Staubli VAL3: start.pgx

program start()
  local num l_nFbkPeriod
  local num l_nMotionPeriod
  local num l_nTrajPeriod
  local num l_nScreenUpdate
  local string l_sVersionMajor
  local num l_nVersionMajor
  local bool l_bOkMajor
  local string l_sVersionMinor
  local num l_nVersionMinor
  local bool l_bOkMinor
begin
  // Copyright (c) 2016, Ocado Technology - Robotics Research Team
  //
  // Licensed under the Apache License, Version 2.0 (the "License");
  // you may not use this file except in compliance with the License.
  // You may obtain a copy of the License at
  //
  //     http://www.apache.org/licenses/LICENSE-2.0
  //
  // Unless required by applicable law or agreed to in writing, software
  // distributed under the License is distributed on an "AS IS" BASIS,
  // WITHOUT WARRANTIES OR CONDITIONS OF ANY KIND, either express or implied.
  // See the License for the specific language governing permissions and
  // limitations under the License.


  // Load interface library for CS8 or CS9
  //
  // CS9 handles the UI differently than CS8, requires
  // the UI funtions to be loaded in seperate libraries

  if(mid(getVersion("System"),1,1) == "7")
    // CS8 - VAL 3 rev 7
    // Check for VAL 3 version >= 7.7
    l_sVersionMajor = mid(getVersion("VAL3"),1,1)
    l_sVersionMinor = mid(getVersion("VAL3"),2,1)
    toNum(l_sVersionMajor, l_nVersionMajor, l_bOkMajor)
    toNum(l_sVersionMinor, l_nVersionMinor, l_bOkMinor)
    if(!l_bOkMajor or !l_bOkMinor)
      popUpMsg("Error reading VAL 3 version")
      taskKill("ros_server~")
    endIf
    if( !((l_nVersionMajor == 7) and (l_nVersionMinor >= 7)))
      // VAL 3 version is too old
      popUpMsg("Error: VAL 3 version is < 7.7, socket communication will not work!")
      taskKill("ros_server~")
    endIf
    libInterface:libLoad("ros_libs/UserInterface/interfaceCS8")
  elseIf(mid(getVersion("System"),1,1) == "8")
    // CS9 - VAL 3 rev 8
    libInterface:libLoad("ros_libs/UserInterface/interfaceCS9")
  endIf

  // feedback task will run every 20ms (50Hz)
  l_nFbkPeriod=0.02
  //l_nFbkPeriod = 0.032 // 30Hz
  //l_nFbkPeriod = 0.05  // 20Hz
  //l_nFbkPeriod = 1.0   //  1Hz

  // motion control task will run every 4ms (250Hz)
  l_nMotionPeriod = 0.004
  //l_nMotionPeriod=0.012  // 83Hz
  //l_nMotionPeriod = 0.05 // 20Hz

  // data (trajectory) reception task will run every 4ms (250Hz)
  l_nTrajPeriod = 0.004
  // not in use at the moment
  l_nScreenUpdate = 1.0

  sStreamTaskName = "streamerTask"
  sTrajPtTaskName = "trajPtTask"
  sMotionTaskName = "motionTask"
  sScreenTaskName = "screenTask"
  sHtbtTaskName = "htbtTask"
  sSystemTaskName = "systemTask"

  // initialise TCP/IP parameters
  call initParams()
  // setup prefix and header of ROS messages
  call setupRosMsgs()

  // socket connection status flags: initially disconnected
  nInConnFlag = 0
  nOutConnFlag = 0
  nSystemConnFlag = 0

  // flag defining whether velocity to be overwritten to max. vel.
  bOverwriteVel = false

  nPtsPopped = 0
  nMovePts = 0

  // flush buffer of incoming socket
  clearBuffer(siTcpIpMotion)
  // flush buffer of outgoing socket
  clearBuffer(siTcpIpFbk)
  // flush buffer of system request socket
  clearBuffer(siTcpIpSystem)

  // check if robot is not in emergency stop and wait until estop is reset
  if(esStatus() == 2)
    popUpMsg("Please reset E-Stop")
    wait(esStatus() < 2)
  endIf

  // before anything else, enable power (only works if robot is in remote mode)
  if(!isPowered())
    if(workingMode() >= 4)
      do
        enablePower()
        delay(2)
      until isPowered()
    else
      popUpMsg("Power must be enabled manually")
    endIf
  endIf

  // reset motion, potentially setting a start joint position for calling autoConnect() in the future
  resetMotion()

  // create joint state and robot status streamer task to send data to industrial_robot_client
  taskCreateSync sStreamTaskName, l_nFbkPeriod, bFbkOverrun, dataStreamer()

  // create trajectory point task to receive data from industrial_robot_client
  taskCreateSync sTrajPtTaskName, l_nTrajPeriod, bTrajPtOverrun, dataReceiver()
  //taskCreate sTrajPtTaskName, 100, dataReceiver()

  // create motion task to synchronously apply motion commands to robot
  taskCreateSync sMotionTaskName, l_nMotionPeriod, bMotionOverrun, motionControl()

  // create synchronous task to update screen
  //taskCreateSync sScreenTaskName, l_nScreenUpdate, bScreenOverrun, screenUpdate()
  taskCreate sScreenTaskName, 10, screenUpdate()

  // create asynchronous task to receive heartbeat on port 11002
  taskCreate sHtbtTaskName, 10, recvHeartbeat()

  // create asynchronous task to handle system requests on port 11001
  taskCreate sSystemTaskName, 100, systemReceiver()

end
